FUNCTION FUN_Divide : REAL
VAR_INPUT
		f_Inp1			: REAL;
		f_Inp2			: REAL;
END_VAR
VAR
END_VAR

IF(f_Inp2 = 0) THEN
	FUN_Divide := 0;
ELSE
	FUN_Divide := f_Inp1 / f_Inp2;
END_IF

END_FUNCTION

(* stored: Version 1.1.0.1, ProductVersion 3.1.4024.9
   POU FUN_Divide: Id {05de8517-1653-41fa-9889-45f8b3cb3ada}, SpecialFunc None *)
